// TwinCAT 3 PLC project IBF_Utilities
// Title: IBF_Utilities
// Company: Industrial Brains B.V.
// ProjectVersion: 2.0.0.0
// Description: Utilities library contains all basic utilities needed like system variables, messages, parameters etc.
// ProgramVersion: 3.1.4022.4
// libraries:
//   Tc2_Standard, * (Beckhoff Automation GmbH)
//   Tc2_System, * (Beckhoff Automation GmbH)
//   Tc2_Utilities, * (Beckhoff Automation GmbH)
//   Tc3_EventLogger, * (Beckhoff Automation GmbH)
//   Tc3_Module, * (Beckhoff Automation GmbH)
// project tree:
//   Avarage/ FB_RollingAverageLREAL.TcPOU (not stored), FB_RollingAverageTime.TcPOU, F_AverageLREAL.TcPOU, F_AverageTime.TcPOU
//   BaseFunctions/ FB_Base.TcPOU, FB_Base_WithEvent.TcPOU (not stored), FB_FunctionBase.TcPOU (not stored), FB_FunctionBase_WIthEvent.TcPOU
//   Compare/Functions/ Between.TcPOU (not stored), Between360deg.TcPOU
//   Conversion/ DegS_To_Rpm.TcPOU, DegS_To_Rpm_And_MMin.TcPOU (not stored), Grey_To_Bin.TcPOU (not stored), MMin_To_Rpm_And_DegS.TcPOU, Rpm_To_DegS.TcPOU (not stored)
//   FaultsAndMessages/Functions/ FB_EventHandler.TcPOU, Fb_FaultHandler.TcPOU (not stored), FB_OperatorMessageDisplay.TcPOU
//   General/DataTypes/ Udt_TimerBandwith.TcDUT (not stored)
//   GVLs/ DataManager.TcGVL (not stored), GVL_FixedValues.TcGVL (not stored), GVL_Message.TcGVL (not stored), GVL_Parameters.TcGVL (not stored), Sys_Variables.TcGVL
//   FaultsAndMessages/DataTypes/ E_ComponentTypes.TcTLEO (not stored), E_Locations.TcTLEO (not stored), E_MessageNumbers.TcTLEO (not stored), E_FaultTypes.TcTLEO, UDT_Fault.TcDUT
//   FaultsAndMessages/ Param_Messages.TcGVL
//   MovePathCalculations/ fAccDecCalc.TcPOU
//   Parameter/DataTypes/Old/ UDT_Parameter_1.TcDUT (not stored), Udt_ParameterRetain.TcDUT (not stored), Udt_Parameter_2.TcDUT (not stored), Udt_ParLog_Old.TcDUT (not stored)
//   Parameter/DataTypes/ Udt_ParameterId.TcDUT (not stored), Udt_Parameter.TcDUT (not stored)
//   Parameter/Functions/ FB_ParameterHandler.TcPOU (not stored), Fb_ParLogging.TcPOU, F_ParToCsvLine.TcPOU
//   PathFunctions/ F_FBNameFromPath.TcPOU, F_GetLevelFromPath.TcPOU (not stored)
//   Positions/FunctionBlocks/ FB_PositionTrigger_Old.TcPOU (not stored), FB_PositionTrigger.TcPOU (not stored)
//   Positions/Functions/ F_AccDecDistanceFromTime.TcPOU, F_AccDecDistanceFromVelo.TcPOU, F_PosCheck.TcPOU (not stored), F_TopVelocityFromTime.TcPOU, F_TriggerPosOffset.TcPOU
//   StepFunctions/ FB_CycleTrigger.TcPOU, FB_Step.TcPOU
//   System/Functions/DataManagement/ FB_PersistentDataManager.TcPOU (not stored)
//   System/Functions/ Fb_SystemVariables.TcPOU (not stored)
//   / Utilities_CD.TcCD (not stored)

// ---- FaultsAndMessages/DataTypes/E_FaultTypes.TcTLEO
{attribute 'qualified_only'}
{attribute 'strict'}
{attribute 'to_string'}
TYPE E_FaultTypes :
(
	NA	:= 0, // Not applicable
	OM 	:= 1, // Operator message
	MC	:= 2, // Missing condition
	CF	:= 3, // Cycle Fault
	FF	:= 4, // Fatal fault
	OW  := 5  // Operator warning
)UDINT;
END_TYPE

// ---- FaultsAndMessages/DataTypes/UDT_Fault.TcDUT
TYPE UDT_Fault :
STRUCT
	// active 
		Active 			: BOOL 				:= FALSE;
	// Message type
 		FaultType 		: E_FaultTypes 		:= E_FaultTypes.NA; // Type of message
	// Message Id number used for translation
		MessageNumber 	: UDINT				:= 0; // message number
		LocationNumber	: UDINT 			:= 0; // message number array ([1]= System, [2]= Module,[3]= sub module, [4]= Component)
	// Message discription
		Discription 	: STRING 			:= ''; // Message text discription in english (service personel only)
	// Location
		LocationName	: STRING			:= ''; // Location discription name
		ComponentType 	: E_ComponentTypes 	:= E_ComponentTypes.NA; // Part type discription
	// Time stamp
		StartTime		: DATE_AND_TIME 	:= DT#2020-1-1-00:00:00 ; // Time and date of message occurence
		EndTime			: DATE_AND_TIME		:= DT#2020-1-1-00:00:00 ; // Time and date of message end
	// Module number
		nModuleID		: UDINT 			; // module reference number used for fault, enable, reset, and safety functions (default := 1, 0 = main system)
	// CompleteFaultnumber for visualization
		FullFaultId		: STRING 			:= 'NA.0.0.0'; // Full fault id for use in HMI is writen by fault function [fault type, message#, location#,ComponentType]
END_STRUCT
END_TYPE

// ---- GVLs/Sys_Variables.TcGVL
(* System variables *)
{attribute 'qualified_only'}
VAR_GLOBAL
// SystemFuntion
	fbSystemVariables : Fb_SystemVariables ;
	AlwaysOn		:BOOL 			;// System variable, Always on bit
	AlwaysOff		:BOOL 			;// System variable, Always off bit
	BlinkFast		:BOOL 			;// System variable, Blink fast bit 1sec 
	BlinkSlow		:BOOL 			;// System variable, Blink slow bit 2 sec
	Pulse1Sec		:BOOL 			;// System variable, Pulse 1 cycle every second
	Pulse100ms		:BOOL 			;// System variable, pulse 1 cycle every 100 ms
	SystemTime		:DT				; // System variable, Windows system time
	TimeZoneId		:E_TimeZoneID 	; // System variable, time zone Id 
	HeartBeat		:BOOL 			;// System Variable, Main system heartbeat 0.5 sec on 0.5 sec off
END_VAR

// ---- FaultsAndMessages/Param_Messages.TcGVL
{attribute 'qualified_only'}
VAR_GLOBAL CONSTANT
	nMAX_MESSAGES_SHOWN 	: UDINT := 10 	;
	nMAX_MESSAGE_HISTORY	: UDINT := 1000 ;
	nMAX_CSV_FIELD_LENGTH	: UDINT := 100	;
	tMESSAGE_TIMEOUT		: TIME 	:= T#5S ;
	sLOGFILE_PATH			: STRING:= 'D:\FaultLogs\'	;
	sLOGFILE_NAME			: STRING:= 'Faultlog' 		; // Message log destination file
	nMESSAGE_COLUMNS		: UDINT := 8 ;
END_VAR

// ---- Avarage/FB_RollingAverageTime.TcPOU
FUNCTION_BLOCK PUBLIC FB_RollingAverageTime
VAR_INPUT
	fInputValue	: TIME ; // Input value [Anny_Number] 
END_VAR
VAR_IN_OUT
	bNewValue		: BOOL ; // Add value to array (set back to false)
	arTimeValues 	: ARRAY [*] OF TIME ; // Array of LREAL values, from thich to get the average
END_VAR
VAR_OUTPUT
	fAverage	: TIME ; // Everage of entries
END_VAR
VAR
	nWriteIndex			: DINT := 0;
	nArrayUpperBound 	: DINT;
	nArrayLowerBound 	: DINT;
	
	reNewValue	: R_TRIG ; // New value trigger
END_VAR

// determine array boundries
nArrayLowerBound := LOWER_BOUND(arTimeValues,1);
nArrayUpperBound := LOWER_BOUND(arTimeValues,1);

// Check if nwrite index is within array bounds
nWriteIndex := LIMIT(nArrayLowerBound, nWriteIndex, nArrayUpperBound);

// Add value to Array 
reNewValue(CLK := bNewValue);
IF reNewValue.Q THEN
	arTimeValues[nWriteIndex] := fInputValue;
	IF nWriteIndex = nArrayUpperBound THEN
		nWriteIndex := nArrayLowerBound;
	ELSE
		nWriteIndex := nWriteIndex +1;
	END_IF
END_IF 

// Calculate average value 
fAverage := F_AverageTime(arTimeValues);

METHOD PUBLIC Cmd_Reset : BOOL
VAR_INPUT
END_VAR
MEMSET(destAddr := ADR(arTimeValues), 0, n := SIZEOF(arTimeValues));
Cmd_Reset := true;
END_METHOD

END_FUNCTION_BLOCK

// ---- Avarage/F_AverageTime.TcPOU
FUNCTION F_AverageTime : TIME
VAR_IN_OUT
	arTimeValues : ARRAY [*] OF TIME ; // Array of LREAL values, from thich to get the average
END_VAR
VAR
	i		: DINT ;
	xSum 	: TIME ; 
	xCount	: DINT ;
END_VAR

FOR i := LOWER_BOUND(arTimeValues,1) TO UPPER_BOUND(arTimeValues,1) DO 
	xSum 	:= arTimeValues[i] + xSum;
	xCount 	:= xCount + 1 ; 
END_FOR

IF xCount >0 THEN 
	F_AverageTime := xSum / xCount;
END_IF

END_FUNCTION

// ---- Avarage/F_AverageLREAL.TcPOU
FUNCTION F_AverageLREAL : LREAL
VAR_IN_OUT
	arLREALValues : ARRAY [*] OF LREAL ; // Array of LREAL values, from thich to get the average
END_VAR
VAR
	i		: DINT ;
	xSum 	: LREAL ; 
	xCount	: DINT ;
END_VAR

FOR i := LOWER_BOUND(arLREALValues,1) TO UPPER_BOUND(arLREALValues,1) DO 
	xSum 	:= arLREALValues[i] + xSum;
	xCount 	:= xCount + 1 ; 
END_FOR

IF xCount >0 THEN 
	F_AverageLREAL := xSum / xCount;
END_IF

END_FUNCTION

// ---- BaseFunctions/FB_Base.TcPOU
FUNCTION_BLOCK PUBLIC ABSTRACT FB_Base
{attribute 'reflection'}
VAR_INPUT
	bEnable			: BOOL 		:= TRUE 	; // Module enable signal reference Default := TRUE (when using system library := GVL_Main.stModules[nModuleId].bEnabled)
	refFbParHandler	: REFERENCE TO Fb_ParLogging 	:= GVL_Parameters.fbParameterHandler	; // reference to parameter handler
	bCmdPause 		: BOOL 		:= FALSE	; // Command Pause functions		
END_VAR
VAR_IN_OUT
	refFbFault	: Fb_FaultHandler	; // reference to fault handler ( when using utilities library := GVL_Main.stModules[nModuleId].fbFaultHandler)
END_VAR
VAR_OUTPUT
	bInitOk			: BOOL 			:= FALSE 	; // function is initialized
	bBussy 			: BOOL 			:= FALSE 	; // device is busy
	bReady			: BOOL 			:= FALSE 	; // device is ready for new command 
	bErrorActive	: BOOL			:= FALSE	; // device Error active 
END_VAR
VAR
	sName			: STRING 		:= ''		; // Name of device distilled from the path 
	nLocationId		: UDINT 		:= 0		; // device id number made up of module and device number				
	
	stFault			: UDT_Fault		; // Fault data from device

	// Function path 
	{attribute 'instance-path'} 
    {attribute 'noinit'}
	sPath			: STRING	; // Path name of function (used for manual reference)
END_VAR

IF __ISVALIDREF(refFbFault) THEN 
	// check if fault is active and send to fault handler
	refFbFault.CmdAddFault(stFault);
END_IF

METHOD PUBLIC CmdReset : BOOL
VAR_INPUT
END_VAR
bErrorActive := FALSE ;

CmdReset := TRUE ;
END_METHOD

METHOD PROTECTED ExecIdentifyDevice : BOOL
VAR_INPUT
	// Message location data
	nId				: UDINT ; // Identification number of object
	nParentId		: UDINT ; // Id of higher level If aplicable (0 = no parent)
	eComponentType	: E_ComponentTypes ; // COmponent or function type for message compilation
END_VAR
// Check device ID
IF nLocationId = 0 THEN
	nLocationId := (nParentId * 10000) + nId * 100 ;
END_IF

// set message location information
stFault.ComponentType 	:= eComponentType;
stFault.LocationName	:= F_FBNameFromPath(sPath := sPath);
stFault.LocationNumber	:= nLocationId ; 

// Get device name from function and add device to manual
IF sName = '' THEN 
	sName := F_FBNameFromPath(sPath := sPath);
END_IF

ExecIdentifyDevice := nLocationId <> 0 AND sName <> '';
END_METHOD

END_FUNCTION_BLOCK

// ---- Parameter/Functions/Fb_ParLogging.TcPOU
FUNCTION_BLOCK PUBLIC Fb_ParLogging EXTENDS FB_ParameterHandler
VAR_OUTPUT
	stParLog		: Udt_ParLog_Old ; // active parameter list
	bReadBusy		: BOOL		:= FALSE	; // File acces Bussy
	bWriteBusy		: BOOL 		:= FALSE	; // file write bussy
	bError			: BOOL		:= FALSE	; // File acces error
	nErrId			: UDINT		:= 0		; // File acces error Id
	nRow	 		: UDINT 	:= 0		;(* Row number (record) *)
	nColumn			: UDINT 	:= 0		;(* Column number (record field) *)
	nInitStep		: UDINT 	:= 0 		; // Initialization step
END_VAR
VAR
	// ====== Compare array =====
		arFileParameters		: ARRAY [1..GVL_Parameters.MAX_PARAMETERS] OF Udt_Parameter;
		nNumberOfParFromFile	: UDINT; // Number of parameters read from file
		nNumberOfChanges		: UDINT; // Number of parameter changes 
		arChangeLog				: ARRAY [0..(GVL_Parameters.MAX_PARAMETERS * 2)] OF STRING ; // Parameter change log 
	// ====== Internal commands ======
		bCmdParFileWrite	: BOOL ; // write alle parameters to .csv file
		bCmdParLogWrite		: BOOL ; // write all changes to .csv file
		bCmdParFileRead		: BOOL ; // Read all parameters from .csv file 
		StParameter			: UDT_Parameter_1 ;
	// ====== File headers ======
		sCsvFileHeader : STRING := 'NUMBER;NAME;TYPE;DISCRIPTION;FACTORY;MAXIMUM;MINIMUM;UNIT;VALUE$L';
	// ====== internal status ======
		bInitOK				: BOOL 	:= FALSE ; // init has been done succesfully
		bFileNotFound		: BOOL 	:= FALSE ; // Parameter file has not been found 
		bParCountDiference	: BOOL 	:= FALSE ; // The number of parameters from file does not match machine 
		bParNumberDiference	: BOOL 	:= FALSE ; // The parameters from file do not match machine
		nDiferenceRow		: UDINT	:= 0	 ; // The file array row number in which diferences were found
 
	// ====== Current step =====
		nReadStep			: INT 	:= 0 	; // File read stepper
		nLogStep			: INT 	:= 0 	; // File logging step
		nWriteStep			: INT 	:= 0 	; // File Write stepper

	// ====== Read variables ======
		hFile				: UINT	:= 0;(* File handle of the source file *)
		cbField				: UDINT	;(* Number of bytes in field buffer *)

	// ====== Read variables ======
		sCSVLine			: T_MaxString := '';(* Single CSV text line (row, record), we are using string as record buffer (your are able to see created fields) *)
		sCSVField			: T_MaxString := '';(* Single CSV field value (column, record field) *)
		sCSVFieldString		: T_MaxString := '';// CSV field converted into string
	// ====== Functions ======
		fbFileOpenForRead	: FB_FileOpen	;(* Opens file *)
		fbFileOpenForWrite	: FB_FileOpen	;(* Opens file *)
		fbFileOpenForLog	: FB_FileOpen	;(* Opens file *)
		fbFileClose			: FB_FileClose	;(* Closes file *)
		fbFileGets			: FB_FileGets	;(* Reads one record (line) *)
		fbFilePuts			: FB_FilePuts	;(* Writes one record (line) *)
		fbReader			: FB_CSVMemBufferReader;(* Helper function block used to parse CSV data bytes (single record line) *)
		fbWriter			: FB_CSVMemBufferWriter;(* Helper function block used to create CSV data bytes (single record line) *)
	
	// Par Read timeout 
		TonParWriteTimeout	: TON := (PT := T#5S) ; // Timeout for parameter read
		TonParreadTimeout	: TON := (PT := T#5S) ; // Timeout for parameter read
		
END_VAR

SUPER^();

// ===== init =====
	IF NOT binitok THEN 
		RETURN;
	ELSE 
		CmdParWriteToFile();
		CmdParLoadFromFile();
	END_IF

METHOD PRIVATE CmdParLoadFromFile : BOOL
VAR_INPUT
END_VAR
VAR 
	i : UDINT ;
	fTempValue	: LREAL ; // Tomporary value to be placed in save value
END_VAR
IF ExecFileRead() THEN 
	;
ELSE
	RETURN;
END_IF

// Compare Parameter counters 
IF nNumberOfParameters <> nNumberOfParFromFile THEN
	bParCountDiference := TRUE ;
ELSE 
	bParCountDiference := FALSE ;
END_IF

// Compare Parameter from file with parameters in machine then write from file to machine
bParNumberDiference := FALSE ;
nDiferenceRow		:= 0 ;
IF NOT bParCountDiference THEN 
	FOR i := 1 TO nNumberOfParameters DO
		IF arParameters[i].nNumber <> arFileParameters[i].nNumber THEN
			bParNumberDiference := TRUE ;
			nDiferenceRow		:= i ;
			CONTINUE;
		ELSE
			IF (arParameters[i].pParameter^.fValue <> arFileParameters[i].fValue) THEN 
				fTempValue := arParameters[i].pParameter^.fValue;  
			ELSE
				fTempValue := 0;
			END_IF
			arParameters[i].pParameter^			:= arFileParameters[i];
			arParameters[i].pParameter^.fSaved 	:= fTempValue;
		END_IF
	END_FOR
END_IF 

CmdParLoadFromFile := TRUE ;
END_METHOD

METHOD PRIVATE CmdParWriteToFile : BOOL
VAR_INPUT
END_VAR
VAR
	i : UDINT ;
	sDTString : STRING ;
END_VAR

IF bCmdParFileWrite THEN 
	FOR i := 1 TO nNumberOfParameters DO
			// Save current actual value for later restore
			IF arParameters[i].pParameter^.fValue <> arFileParameters[i].fValue THEN
				arParameters[i].pParameter^.fSaved := arFileParameters[i].fValue ;
			END_IF
			arFileParameters[i] := arParameters[i].pParameter^ ;
	END_FOR
END_IF

//IF nNumberOfChanges > 0 AND NOT bParCountDiference THEN 
//	ExecWriteToLog();
//END_IF
CmdParWriteToFile := ExecFileWrite();
END_METHOD

METHOD PUBLIC CmdSavePar : BOOL
VAR_INPUT
END_VAR
bCmdParFileWrite := TRUE ;

CmdSavePar := bWriteBusy ;
END_METHOD

METHOD PRIVATE ExecFileRead : BOOL
VAR_INPUT
END_VAR
VAR
	i : UDINT := 0 ;
END_VAR
// ===== Wait for command =====
	IF bCmdParFileRead OR bReadBusy THEN 
		;
	ELSE
		RETURN ;
	END_IF

// ===== prepare for file read =====
	CASE nReadStep OF
		0:	(* Wait for rising edge at bRead variable *)
			bReadBusy		:= TRUE;
			bFileNotFound	:= FALSE ;
			bCmdParFileRead := FALSE ;
			bError			:= FALSE;
			nErrId			:= 0;
			hFile			:= 0;
			nRow			:= 0;
			nColumn			:= 0;
			nReadStep 			:= 1;
	
		1:	(* Open source file *)
			fbFileOpenForRead(  bExecute := FALSE  );
			fbFileOpenForRead( sNetId := GVL_Parameters.sNetId, sPathName := GVL_Parameters.sPARLIST_FILE, nMode := FOPEN_MODEREAD OR FOPEN_MODETEXT,(* Open file in text mode! *)
						ePath := PATH_GENERIC, bExecute := TRUE );
			nReadStep := 2;
	
		2:(* Wait until open not busy *)
			fbFileOpenForRead( bExecute := FALSE, bError => bError, nErrID => nErrID, hFile => hFile );
			IF NOT fbFileOpenForRead.bBusy THEN
				IF NOT fbFileOpenForRead.bError THEN
					nReadStep := 3;
				ELSE(* Error: file not found? *)
					bFileNotFound := TRUE ;
					nReadStep := 100;
				END_IF
			END_IF
		3:	(* Read single line (record) *)
			fbFileGets( bExecute := FALSE );
			fbFileGets( sNetId := GVL_Parameters.sNetId, hFile := hFile, bExecute := TRUE );
			nReadStep := 4;
		4:(* Wait until read not busy *)
			fbFileGets( bExecute := FALSE, bError => bError, nErrID => nErrID, sLine => sCSVLine );
			IF NOT fbFileGets.bBusy THEN
				IF NOT fbFileGets.bError THEN
					IF fbFileGets.bEOF THEN
						nReadStep 				:= 10;(* End of file reached => Close source file *)
					ELSE
						(* FB_FileGets returns text line without the CR (carriage return) character.
						We have to restore the CR character (replace the $L character with $R$L characters) *)
						IF RIGHT( sCSVLine, 1 ) = '$L' THEN
							sCSVLine := REPLACE( sCSVLine, '$R$L', 2, LEN( sCSVLine ) );
						END_IF
						nReadStep := 5;
					END_IF
				ELSE(* Error *)
					nReadStep := 100;
				END_IF
			END_IF
		5:(* Parse single line (record) *)
			fbReader.eCmd := eEnumCmd_First;(* Read first field value *)
			REPEAT
				fbReader( pBuffer := ADR( sCSVLine ), cbBuffer := SIZEOF( sCSVLine ), getValue => sCSVField );
				IF fbReader.bOk THEN
					fbReader.eCmd := eEnumCmd_Next;(* Read next field value *)
					IF ( nRow <= GVL_Parameters.MAX_PARAMETERS ) AND nRow > 0 THEN
						IF ( nColumn <= GVL_Parameters.PAR_COLUMNS ) THEN
							sCSVFieldString	:= CSVFIELD_TO_STRING( sCSVField, TRUE);
							CASE nColumn OF
									0: // Parameter number [Udint]	
										arFileParameters[nRow].nNumber		:= STRING_TO_UDINT(sCSVFieldString); 						
									1: // Parameter Name [string]
										arFileParameters[nRow].sName 		:= sCSVFieldString;							
									2: // Parameter type [String]
										arFileParameters[nRow].sType 		:= sCSVFieldString;	
									3: // Parameter discription [string]
										arFileParameters[nRow].sDiscription	:= sCSVFieldString;						
									4: // Parameter factory value [LREAL]
										arFileParameters[nRow].fFactory		:= STRING_TO_LREAL(sCSVFieldString);							
									5: // Parameter maximum value [LREAL]
										arFileParameters[nRow].fMaximum		:= STRING_TO_LREAL(sCSVFieldString);							
									6: // Parameter minimum value[LREAL]
										arFileParameters[nRow].fMinimum		:= STRING_TO_LREAL(sCSVFieldString);							
									7: // Parameter unit {String]
										arFileParameters[nRow].sUnit 		:= sCSVFieldString;							
									8: // Parameter value [LREAL]
										arFileParameters[nRow].fValue		:= STRING_TO_LREAL(sCSVFieldString);							
							ELSE
								;
							END_CASE
							nColumn := nColumn + 1;(* Increment number of read columns *)
						END_IF
					END_IF
					IF fbReader.bCRLF THEN(* CRLF == TRUE => End of reacord reached *)
						nNumberOfParFromFile := nRow;
						nRow 		:= nRow + 1;(* Increment number of read records *)
						nColumn 	:= 0;(* Reset number of columns *)
					END_IF
				ELSE(* Error: End of record reached or all fields read *)
					nReadStep := 3;(* Try to read next line *)
				END_IF
			UNTIL NOT fbReader.bOk
			END_REPEAT
		10:	(* Close source file *)
			fbFileClose( bExecute := FALSE );
			fbFileClose( sNetId := GVL_Parameters.sNetId, hFile := hFile, bExecute := TRUE );
			nReadStep := 11;
	
		11:(* Wait until close not busy *)
			fbFileClose( bExecute := FALSE, bError => bError, nErrID => nErrID );
			IF ( NOT fbFileClose.bBusy ) THEN
				hFile := 0;
				nReadStep := 100;
			END_IF
		100: (* Error or ready nReadStep => cleanup *)
			IF ( hFile <> 0 ) THEN
				nReadStep := 10; (* Close the source file *)
			ELSE
				bReadBusy := FALSE;
				ExecFileRead := TRUE ;
				nReadStep := 0;	(* Ready *)
			END_IF
	END_CASE
	
	TonParreadTimeout(IN := bReadBusy);
	bError S= TonParreadTimeout.Q;
END_METHOD

METHOD INTERNAL ExecFileWrite : BOOL
VAR_INPUT
END_VAR
// ===== Wait for command =====
	IF bCmdParFileWrite OR bWriteBusy THEN 
		;
	ELSE
		RETURN ;
	END_IF

// ===== Start file write =====
	CASE nWriteStep OF
		0:	(* Wait for rising edge at bWrite variable *)
				bFileNotFound		:= FALSE ;
				bParCountDiference	:= FALSE ;
				bWriteBusy 			:= TRUE;
				bCmdParFileWrite	:= FALSE ;
				bError				:= FALSE;
				nErrId				:= 0;
				hFile				:= 0;
				nRow				:= 0;
				nWriteStep 				:= 1;
		1:	(* Open source file *)
			fbFileOpenForWrite(  bExecute := FALSE  );
			fbFileOpenForWrite( sNetId := GVL_Parameters.sNetId, sPathName := GVL_Parameters.sPARLIST_FILE, nMode := FOPEN_MODEWRITE OR FOPEN_MODETEXT,(* Open file in TEXT mode! *)
						ePath := PATH_GENERIC, bExecute := TRUE );
			nWriteStep := 2;
		2:(* Wait until open not busy *)
			fbFileOpenForWrite( bExecute := FALSE, bError => bError, nErrID => nErrID, hFile => hFile );
			IF NOT fbFileOpenForWrite.bBusy THEN
				IF NOT fbFileOpenForWrite.bError THEN
					nWriteStep := 3;
				ELSE(* Error: file not found? *)
					nWriteStep := 100;
				END_IF
			END_IF
	
		3:(* Convert one PLC parameter field to CSV format *)
			// Go column by column to avoid return strings that are too long
			// TODO test (default string constructor is 80 characters, but can be extended to <?>)
			IF nRow = 0 THEN 
				sCSVLine := sCsvFileHeader;
			ELSE
				sCSVLine := F_ParToCsvLine(stParameter := arFileParameters[nRow], nColumn := nColumn);
			END_IF
			nWriteStep := 4 ;
		4:	(* Write single Field *)
			fbFilePuts( bExecute := FALSE );
			fbFilePuts( sNetId := GVL_Parameters.sNetId, hFile := hFile, sLine := sCSVLine, bExecute := TRUE );
			nWriteStep := 5;
		5:(* Wait until write not busy *)
			fbFilePuts( bExecute := FALSE, bError => bError, nErrID => nErrID );
			IF NOT fbFilePuts.bBusy THEN
				IF NOT fbFilePuts.bError THEN
					nWriteStep := 3;(* Write next record *)
					IF nRow = 0 OR nColumn = 8 THEN
						nColumn := 0 ;
						nRow := nRow + 1;
						IF nRow = nNumberOfParameters + 1 THEN
							nWriteStep := 10;
						END_IF;
					ELSE
						nColumn := nColumn + 1;
					END_IF
				ELSE(* Error *)
					nWriteStep := 100;
				END_IF
			END_IF
		10:	(* Close source file *)
			fbFileClose( bExecute := FALSE );
			fbFileClose( sNetId := GVL_Parameters.sNetId, hFile := hFile, bExecute := TRUE );
			nWriteStep := 11;
	
		11:(* Wait until close not busy *)
			fbFileClose( bExecute := FALSE, bError => bError, nErrID => nErrID );
			IF ( NOT fbFileClose.bBusy ) THEN
				hFile := 0;
				nWriteStep := 100;
			END_IF
	
		100: (* Error or ready nWriteStep => cleanup *)
			IF ( hFile <> 0 ) THEN
				nWriteStep := 10; (* Close the source file *)
			ELSE
				bParCountDiference 	:= FALSE ;
				bWriteBusy 			:= FALSE;
				ExecFileWrite		:= TRUE ;
				nWriteStep 			:= 0;	(* Ready *)
			END_IF
	
	END_CASE
	
	TonParWriteTimeout(IN := bWriteBusy);
	bError	S= TonParWriteTimeout.Q ;
	

ExecFileWrite := TRUE ;
END_METHOD

METHOD PRIVATE ExecWriteToLog : BOOL
VAR_INPUT
END_VAR
VAR
	sTempField : STRING ;
END_VAR
// ===== Wait for command =====
	IF bWriteBusy OR bCmdParLogWrite THEN 
		;
	ELSE
		RETURN ;
	END_IF

// ===== Start file write =====
CASE nLogStep OF
	0:	(* Wait for rising edge at bWrite variable *)
			bWriteBusy 			:= TRUE;
			bCmdParLogWrite	:= FALSE ;
			bError				:= FALSE;
			nErrId				:= 0;
			hFile				:= 0;
			nRow				:= nNumberOfChanges * 2; // Twice the number of changes because old and new values are stored sequentially in teh same array
			nLogStep 			:= 1;
	1:	(* Open source file *)
		fbFileOpenForLog(  bExecute := FALSE  );
		fbFileOpenForLog( sNetId := GVL_Parameters.sNetId, sPathName := GVL_Parameters.sPARLIST_FILE, nMode := FOPEN_MODETEXT,(* Open file in TEXT mode! *)
					ePath := PATH_GENERIC, bExecute := TRUE );
		nLogStep := 2;
	2:(* Wait until open not busy *)
		fbFileOpenForLog( bExecute := FALSE, bError => bError, nErrID => nErrID, hFile => hFile );
		IF NOT fbFileOpenForLog.bBusy THEN
			IF NOT fbFileOpenForLog.bError THEN
				nLogStep := 3;
			ELSE(* Error: file not found? *)
				nLogStep := 100;
			END_IF
		END_IF

	3:(* Convert one PLC record to CSV format *)
		sCSVLine := arChangeLog[nRow];
		nLogStep := 4 ;
	4:	(* Write single text line *)
		fbFilePuts( bExecute := FALSE );
		fbFilePuts( sNetId := GVL_Parameters.sNetId, hFile := hFile, sLine := sCSVLine, bExecute := TRUE );
		nLogStep := 5;

	5:(* Wait until write not busy *)
		fbFilePuts( bExecute := FALSE, bError => bError, nErrID => nErrID );
		IF NOT fbFilePuts.bBusy THEN
			IF nRow = 0 THEN
				nNumberOfChanges := 0;
				nLogStep := 10;
			ELSIF NOT fbFilePuts.bError THEN
				arChangeLog[nRow] := ''; // Delete change from log
				nRow := nRow - 1;
				nLogStep := 3;(* Write next record *)
			ELSE(* Error *)
				nLogStep := 100;
			END_IF
		END_IF
	10:	(* Close source file *)
		fbFileClose( bExecute := FALSE );
		fbFileClose( sNetId := GVL_Parameters.sNetId, hFile := hFile, bExecute := TRUE );
		nLogStep := 11;

	11:(* Wait until close not busy *)
		fbFileClose( bExecute := FALSE, bError => bError, nErrID => nErrID );
		IF ( NOT fbFileClose.bBusy ) THEN
			hFile := 0;
			nLogStep := 100;
		END_IF

	100: (* Error or ready nLogStep => cleanup *)
		IF ( hFile <> 0 ) THEN
			nLogStep := 10; (* Close the source file *)
		ELSE
			bWriteBusy := FALSE;
			nLogStep := 0;	(* Ready *)
		END_IF
END_CASE
END_METHOD

METHOD PUBLIC Init : BOOL
VAR_INPUT
END_VAR
// Read parameters from .CSV file and check if load is valid

CASE nInitStep OF 
	0: //check if init has been done 
		bInitOK 	:= FALSE;
		nInitStep 	:= 10 ;
	10: // start File read
		bCmdParFileRead := TRUE ;
		nInitStep := 11; 
	11: // Execute file read 
		IF CmdParLoadFromFile() THEN 
			nInitStep := 12 ;
		END_IF
	12: // Check if read is valid 
		IF bFileNotFound OR bParCountDiference THEN 
			nInitStep := 20 ;
		ELSE 
			nInitStep := 100 ;
		END_IF
	20: // start File write
		bCmdParFileWrite:= TRUE ;
		nInitStep		:= 21 ;
	21: // Wait for file write to finish
		IF CmdParWriteToFile() THEN 
			nInitStep := 100 ;
		ELSIF bError THEN 
			nInitStep := 900 ; 
		END_IF 
	100: // Init ok 
		bInitOK 	:= TRUE ;
		Init		:= TRUE ;
		nInitStep	:= 0 ;
	900: // file fault	
		bInitOK := FALSE ;
		RETURN ;
	ELSE 
		;
END_CASE
END_METHOD

END_FUNCTION_BLOCK

// ---- Parameter/Functions/F_ParToCsvLine.TcPOU
FUNCTION F_ParToCsvLine : T_MaxString // convert parameter into csv string (default UDt_Parameter setup)
VAR_INPUT
	stParameter : Udt_Parameter ; 
	nColumn		: UDINT ;
END_VAR
VAR
	sTempString : T_MaxString;
	sTempCsvField : T_MaxString;
END_VAR

CASE nColumn OF 
	0: // number
		sTempString := UDINT_TO_STRING(stParameter.nNumber);
	1: // name
		sTempString := stParameter.sName;
	2: // Type
		sTempString := stParameter.sType;
	3: // discription
		sTempString := stParameter.sDiscription;
	4: // factory
		sTempString := LREAL_TO_STRING(stParameter.fFactory);
	5: // maximum
		sTempString := LREAL_TO_STRING(stParameter.fMaximum);
	6: // minimum
		sTempString := LREAL_TO_STRING(stParameter.fMinimum);
	7: // Unit 
		sTempString := stParameter.sUnit;
	8: // value
		sTempString := LREAL_TO_STRING(stParameter.fValue);
	ELSE
		;
END_CASE

sTempCsvField := STRING_TO_CSVFIELD(sTempString, FALSE);
IF nColumn < 8 THEN 
	sTempCsvField := CONCAT(StempCsvField,';');
ELSE
	sTempCsvField := CONCAT(StempCsvField,'$L');
END_IF

F_ParToCsvLine := sTempCsvField;

END_FUNCTION

// ---- PathFunctions/F_FBNameFromPath.TcPOU
FUNCTION F_FBNameFromPath : STRING // distills .fb name from function path
VAR_INPUT
	sPath	: STRING ;
END_VAR
VAR
	sTemp		: STRING ;
	nstartFbName: INT ; 
END_VAR

sTemp := sPath ;

REPEAT 
	// Look for first occurance of .fb in string
	nStartFbName := FIND( sTemp,'.fb');
	// Delete text before .fb and .fb itself
	IF nstartFbName <>0 THEN 
		sTemp := DELETE( STR := sTemp, LEN := nstartFbName + 3, 0); 
	END_IF
UNTIL
	nstartFbName = 0 
END_REPEAT

F_FBNameFromPath := sTemp ;

END_FUNCTION

// ---- BaseFunctions/FB_FunctionBase_WIthEvent.TcPOU
{attribute 'reflection'}
FUNCTION_BLOCK PUBLIC ABSTRACT FB_FunctionBase_WIthEvent EXTENDS FB_Base_WithEvent
VAR_INPUT
	bSafetyOk	: BOOL 		:= TRUE 				; // Module can operate safely [default true]
END_VAR
VAR_OUTPUT
	sActiveState	: STRING 		:= 'Idle'	; // active state of device 
	bManual			: BOOL 			:= FALSE 	; // device is in manual mode
	bIsSafe			: BOOL 			:= FALSE	; // Device is locked and safe
	bHeld			: BOOL 			:= FALSE 	; // Function is held
	bBlockedCommand	: BOOL 			:= FALSE 	; // a device command is blocked because of collision detect 
END_VAR
VAR
	bCmdManual 		: BOOL			:= FALSE	; // manual commands enabled control functions (thus disable automatic)
END_VAR

SUPER^();

// Communicate active state
IF NOT bSafetyOk THEN 
	sActiveState := 'Safety not ok';
ELSIF bErrorActive THEN 
	sActiveState := 'Error is active';
ELSIF NOT bInitOk THEN 
	sActiveState := 'Not initialized';
ELSIF bManual THEN 
	sActiveState := 'Operational';
END_IF 

// check for manual command mode
bManual := bCmdManual ;

// Execute device functions
IF bInitOk THEN  
	ExecMachineSafety();
	ExecDevFunctions();
END_IF

// Set fault if commands are blocked
IF bBlockedCommand THEN 
	fbEvent.CmdAddEvent( Event := TC_EVENTS.StateMessages.FunctionsIsBlocked);
END_IF

METHOD PUBLIC CmdHold : BOOL
VAR_INPUT
END_VAR
bHeld 	:= TRUE ;
CmdHold := bHeld ;
END_METHOD

METHOD PUBLIC CmdManual : BOOL
VAR_INPUT
END_VAR
bCmdManual := true ;
END_METHOD

METHOD PUBLIC CmdSafeStop : BOOL
VAR_INPUT
END_VAR
// check if device is safe
bIsSafe 	:= NOT bEnable ;
CmdSafeStop := bIsSafe ;
END_METHOD

METHOD PROTECTED ExecDevFunctions : BOOL
VAR_INPUT
END_VAR
END_METHOD

METHOD PROTECTED ExecMachineSafety : BOOL
VAR_INPUT
END_VAR
END_METHOD

END_FUNCTION_BLOCK

// ---- Compare/Functions/Between360deg.TcPOU
FUNCTION Between360deg : BOOL // Returns true if value is >= the lower and <= the upper threshold, if lower > upper then upper := Upper +360 deg
VAR_INPUT
	Lower	: LREAL	; // lower threshold value [LREAL]
	Value	: LREAL	; // test value [LREAL]
	Upper	: LREAL	; // Upper threshold value [LREAL]
END_VAR
VAR
END_VAR

IF Lower > Upper THEN  
	Between360deg S= Between( Lower, Value, 360);
	Between360deg S= Between( 0, Value, Upper)	;
ELSE 
	Between360deg S= Between( Lower, Value, Upper)	;
END_IF

END_FUNCTION

// ---- Conversion/DegS_To_Rpm.TcPOU
(* convert degrees per second to rotations per minute *)
FUNCTION DegS_To_Rpm : LREAL
VAR_INPUT
	DegS : LREAL ; // Input degrees per second as long real
END_VAR

// ===== convert degrees per second to Rpm =====
	DegS_To_Rpm := (DegS/360)*60 ;

END_FUNCTION

// ---- Conversion/MMin_To_Rpm_And_DegS.TcPOU
(* Convert meters per minute to degrees per second *)
FUNCTION MMin_To_Rpm_And_DegS : BOOL
VAR_INPUT
	MeterPerMinute 	: LREAL ; // Input meters per minute
	StitchLength	: LREAL ; // Input Stitch length
END_VAR
VAR_OUTPUT
	RevPerMinute	: LREAL ; // Output revolutions per minute
	DegPerSecond	: LREAL ; // Output degrees per second
END_VAR
VAR
	MmMin 	: LREAL ; // Millimeters per minute
	RevSec 	: LREAL ; // Millimeters per second
END_VAR

// ===== convert MMin to RPM =====
	RevPerMinute := (MeterPerMinute * 1000) / StitchLength ;
//===== Convert RPM to DegS =====
	DegPerSecond := (RevPerMinute/60)*360 ;

END_FUNCTION

// ---- FaultsAndMessages/Functions/FB_EventHandler.TcPOU
FUNCTION_BLOCK PUBLIC FB_EventHandler
VAR_INPUT
	nTwincErrorId	: UDINT := 0; // OPTIONAL Error Id from twincat function block library
END_VAR
VAR_OUTPUT
	// Active events
	bActOM 			: BOOL := FALSE ;
	bActMC 			: BOOL := FALSE ;
	bActCF 			: BOOL := FALSE ;
	bActFF 			: BOOL := FALSE ;
	// Last event
	stLastEvent		: TcEventEntry 	; // Event entry discription  
END_VAR
VAR // Event Conformation data
	bConfRequired 	: BOOL := FALSE ; // Conformation of  		
	// Resetting
	bResetting		: BOOL := FALSE ;
END_VAR
VAR // location data
	// Location
	nLocationNumber	: UDINT 			:= 0; // message number array ([1]= System, [2]= Module,[3]= sub module, [4]= Component)
	sLocationName	: STRING			:= ''; // Location discription name
	eComponentType 	: E_ComponentTypes 	:= E_ComponentTypes.NA; // Part type discription
	// Module number
	nModuleID		: UDINT 			; // module reference number used for fault, enable, reset, and safety functions (default := 1, 0 = main system)
	// Source
	fbSource		: FB_TcSourceInfo;
END_VAR
VAR // Event functions 
	fbAlarm		: FB_TcAlarm ; // alarm event function
	fbMessage 	: FB_TcMessage ; // Message event
	
	hr 			: HRESULT;
	hrLastError : HRESULT;
END_VAR

METHOD PUBLIC CmdAddEvent : BOOL
VAR_INPUT
	Event			: TcEventEntry ; // Event entry discription  
END_VAR
// check if allarm has already been raised
IF fbAlarm.EqualsToEventEntryEx(stOther	:= Event) THEN
	CmdAddEvent := TRUE;
	RETURN;
END_IF

// Check Event severity
CASE Event.eSeverity OF 
	TcEventSeverity.Critical:
		bActFF 			S= TRUE ;	
		fbAlarm.CreateEx(Event,TRUE,fbSource);
		hr := fbAlarm.Raise(0);
	TcEventSeverity.Error:
		bActCF 			S= TRUE ;	
		fbAlarm.CreateEx(Event,TRUE,fbSource);
		hr := fbAlarm.Raise(0);
	TcEventSeverity.Warning:
		bActMC 			S= TRUE ;	
		fbAlarm.CreateEx(Event,FALSE,fbSource);
		hr := fbAlarm.Raise(0);
	TcEventSeverity.Info:
		bActOM 			S= TRUE ;	
		fbMessage.CreateEx(Event,fbSource);
		hr := fbMessage.Send(0);
	ELSE 
		RETURN;
END_CASE

// Add aditional error id
IF nTwincErrorId >0 THEN 
	fbAlarm.ipArguments.AddUDInt( value := nTwincErrorId);
END_IF
nTwincErrorId := 0; // Always clear error id after check

IF FAILED(hr) THEN 
	hrLastError := hr ;
ELSE
	CmdAddEvent := TRUE;
END_IF
END_METHOD

METHOD PUBLIC CmdReset : BOOL
VAR_INPUT
END_VAR
bResetting := TRUE ;

hr := fbAlarm.Clear(0,TRUE);

IF NOT FAILED(hr) THEN 
	bResetting := FALSE ; 
	bActOM 	:= FALSE ;
	bActMC	:= FALSE ;
	bActCF	:= FALSE ;
	bActFF	:= FALSE ;
END_IF

// Set feedback
CmdReset := NOT bResetting;
END_METHOD

METHOD PRIVATE ExecSetActiveEvents : BOOL
VAR_INPUT
END_VAR
END_METHOD

METHOD PUBLIC Init : BOOL
VAR_INPUT
	// Location
		sLocationName	: STRING			:= ''; // Location discription name
		eComponentType 	: E_ComponentTypes 	:= E_ComponentTypes.NA; // Part type discription
	// Module number
		nModuleID		: UDINT 			; // module reference number used for fault, enable, reset, and safety functions (default := 1, 0 = main system)
END_VAR
// Transfer location data into event location data format
fbSource.nId 	:= nModuleID;
fbSource.sName	:= TO_STRING(eComponentType);
fbSource.ExtendName(sLocationName);

fbMessage.CreateEx(TC_EVENTS.StateMessages.ModuleInitialized,fbSource);
fbMessage.Send(0);

Init := TRUE ;
END_METHOD

END_FUNCTION_BLOCK

// ---- FaultsAndMessages/Functions/FB_OperatorMessageDisplay.TcPOU
FUNCTION_BLOCK FB_OperatorMessageDisplay // function compares messages and shows latest message on screen for a set period of time
VAR_INPUT
	bEnable 	: BOOL 	:= TRUE ; // enable messages
	tDisplayTime: TIME	:= Param_Messages.tMESSAGE_TIMEOUT ; // Time before message relevance is checked (default = Param_Messages.tMESSAGE_TIMEOUT)
END_VAR
VAR_IN_OUT
	sMessage 	: STRING ; // Operator message (default = GVL_Message.sOPeratorMessage)
END_VAR
VAR_OUTPUT
	sOutMessage : STRING ; // message output to screen
END_VAR
VAR
	sOldMessage 	: STRING := ''; // old message as displayed 
	tonDisplayTimer	: TON ; // Display timer
END_VAR

// Run timers
tonDisplayTimer(PT := tDisplayTime);

// compare old message with new message 
IF sMessage = sOldMessage THEN 
	tonDisplayTimer.IN := TRUE ;
	IF tonDisplayTimer.Q = TRUE THEN 
		sMessage := '';
	END_IF
ELSE 
	tonDisplayTimer.IN 	:= FALSE 	;
	sOldMessage 		:= sMessage ; 
END_IF

// write message to display
sOutMessage := sMessage ;

END_FUNCTION_BLOCK

// ---- MovePathCalculations/fAccDecCalc.TcPOU
FUNCTION fAccDecCalc : LREAL // calculates acceleration and deceleration values from path [units/sec^2]
VAR_INPUT
	fVelocity		: LREAL ; // current velocity [units]
	fNewVelocity	: LREAL ; // New velocity [units] 
	fDistance		: LREAL ; // Travel distance [units]
END_VAR
VAR
	xDeltaVelo		: LREAL ; // delta velocity
	xAverageVelo	: LREAL ; // Average velocity
	xTime			: LREAL ; // Time it takes to slow down [s]
END_VAR

xDeltaVelo	:= ABS(fVelocity - fNewVelocity);
xAverageVelo:= ABS(fVelocity + fNewVelocity)/2;
xTime		:= fDistance / xAverageVelo ;
fAccDecCalc	:= xDeltaVelo / xTime ;

END_FUNCTION

// ---- Positions/Functions/F_AccDecDistanceFromTime.TcPOU
FUNCTION F_AccDecDistanceFromTime : LREAL
VAR_INPUT
	nAccelDecel	: LREAL ; // acceleration or deceleration [units/s^2]
	nTimeMs		: LREAL	; // Time for acceleratio/ deceleration to take place [ms]
END_VAR
VAR
	nTimeSec	: LREAL;
	nVelocity	: LREAL;
END_VAR

nTimeSec := nTimeMs/1000;

nVelocity := nAccelDecel * nTimeSec;

F_AccDecDistanceFromTime := nVelocity * nTimeSec / 2 ;

END_FUNCTION

// ---- Positions/Functions/F_AccDecDistanceFromVelo.TcPOU
FUNCTION F_AccDecDistanceFromVelo : LREAL
VAR_INPUT
	nVelocity	: LREAL ; // velocity [m/s]
	nAccDecc	: LREAL ; // acceleration or deceleration value [m/s^2]
END_VAR
VAR
	nTime : LREAL ;
END_VAR

nTime := nVelocity	/	nAccDecc ;

F_AccDecDistanceFromVelo := nVelocity * (nTime/2);

END_FUNCTION

// ---- Positions/Functions/F_TopVelocityFromTime.TcPOU
FUNCTION F_TopVelocityFromTime : LREAL
VAR_INPUT
	nAccel	: LREAL ; // acceleration or deceleration [units/s^2]
	nTimeMs		: LREAL	; // Time for acceleratio/ deceleration to take place [ms]
END_VAR
VAR
	nTimeSec	: LREAL;
END_VAR

nTimeSec := nTimeMs/1000;

F_TopVelocityFromTime := nAccel * nTimeSec;

END_FUNCTION

// ---- Positions/Functions/F_TriggerPosOffset.TcPOU
(* function to calculate trigger points for time based moves *)
FUNCTION F_TriggerPosOffset : LREAL
VAR_INPUT
	Velocity		: LREAL	; // [Units/sec] command velocity 
	nMoveTimeMs		: LREAL	; // [ms] Time it takes for move to complete
END_VAR
VAR
END_VAR

// ===== Convert time to usable calculation value =====
	F_TriggerPosOffset := nMovetimeMs * ABS(Velocity / 1000);

END_FUNCTION

// ---- StepFunctions/FB_CycleTrigger.TcPOU
FUNCTION_BLOCK FB_CycleTrigger // This function can be used to start state machines and wait for them to finish
VAR_OUTPUT
	bStart 	: BOOL ; // Start cycle 
	bBusy 	: BOOL ; // cycle is bussy
	bDone	: BOOL ; // cycle is done
END_VAR
VAR
	fbreStartCycle : R_TRIG ; // rising edge trigger for cycle start
END_VAR

ACTION Reset:
bDone 	:= FALSE;
bBusy 	:= FALSE;
bStart	:= FALSE;
END_ACTION

ACTION SetDone:
bBusy := FALSE 	;
bDone := TRUE	;
END_ACTION

ACTION SetStart:
IF fbreStartCycle.Q THEN
	bBusy := TRUE; 
ELSIF bDone THEN 
	bStart := FALSE;
ELSE
	bStart := TRUE;
END_IF

fbreStartCycle(CLK := bStart);
END_ACTION

END_FUNCTION_BLOCK

// ---- StepFunctions/FB_Step.TcPOU
FUNCTION_BLOCK PUBLIC FB_Step EXTENDS FB_Base
VAR_INPUT
END_VAR
VAR_OUTPUT
	nActStep	: UDINT := 0 ; // Active step
	bIdle		: BOOL	:= TRUE  ; // Stepper is idle (Step 0)
	bPaused		: BOOL 	:= FALSE ; // Stepper is paused
	bHold		: BOOL 	:= FALSE ; // Stepper is blocked for changes
	bSkipPause	: BOOL	:= FALSE ; // Pause function is skipped in this step 
	bResetting	: BOOL  := False ; // Reset is active
END_VAR
VAR
	nPreviousStep 	: UDINT ; // Previous active step
	nNextStep		: UDINT ; // Next step to activate
	nResetStep		: UDINT ; // step to which the stepper will go after reset
END_VAR

SetActiveStep();

METHOD PUBLIC CmdHold : BOOL
VAR_INPUT
END_VAR
bHold := TRUE ;

CmdHold := bHold;
END_METHOD

METHOD PUBLIC CmdNext : BOOL
VAR_INPUT
END_VAR
IF NOT bHold THEN 
	nNextStep := nActStep +	1 ;	
END_IF

CmdNext := TRUE ;
END_METHOD

METHOD PUBLIC CmdPrevious : BOOL
VAR_INPUT
END_VAR
IF NOT bHold THEN 
	nNextStep := nPreviousStep ;	
END_IF

CmdPrevious := TRUE ;
END_METHOD

METHOD PUBLIC CmdReset : BOOL
VAR_INPUT
END_VAR
bErrorActive := FALSE ;

IF nActStep <> nResetStep THEN 
	IF NOT bResetting THEN
		bResetting := TRUE ;
	ELSE
		nPreviousStep 	:= nActStep ;
		nNextStep		:= nResetStep ;
		nActStep 		:= nResetStep ;
		bResetting 		:= FALSE;
	END_IF
ELSE
	CmdReset := TRUE ; 
END_IF
END_METHOD

METHOD PUBLIC CmdToStep : BOOL
VAR_INPUT
	nStep	: UDINT ;
END_VAR
IF NOT bHold THEN 
	nNextStep := nStep ;
END_IF

CmdToStep := nNextStep = nStep ;
END_METHOD

METHOD PUBLIC Init : BOOL
VAR_INPUT
	// Location data for messages  
	nId			: UDINT ; // Identification number of object
	nParentId	: UDINT ; // Id of higher level If aplicable (0 = no parent)
	nResetStep	: UDINT ; // step to which the stepper wil go at reset
END_VAR
// ====== Calculate device id =====
	ExecIdentifyDevice(nId,nParentId,E_ComponentTypes.StepProgram);
	
// ===== set reset step ======
	nActStep 			:= nResetStep ;
	THIS^.nResetStep	:= nResetStep ;
END_METHOD

METHOD PRIVATE SetActiveStep : BOOL
VAR_INPUT
END_VAR
IF bResetting THEN 
	nPreviousStep 	:= nActStep ;
	nNextStep		:= nResetStep ;
	nActStep 		:= nResetStep ;
	bResetting 		:= FALSE; 
ELSIF bHold THEN 
	bHold 			:= FALSE ;
	RETURN; 
ELSIF bErrorActive THEN 
	stFault.Active			:= TRUE ;
	stFault.ComponentType	:= E_ComponentTypes.StepProgram ;
	stFault.Discription		:= CONCAT(sName, ' Invalid step state');
	stFault.FaultType		:= E_FaultTypes.FF;
	stFault.MessageNumber	:= E_MessageNumbers.FF_ComunicationFault;
ELSIF NOT bCmdPause OR bSkipPause THEN 
	IF nActStep <> nNextStep THEN 
		nPreviousStep 	:=	nActStep;	
		nActStep		:= 	nNextStep;
	END_IF
END_IF

bPaused 	:= bCmdPause ;	
bSkipPause 	:= FALSE ; 
bIdle 		:= nActStep = 0 ;
END_METHOD

METHOD Public SkipPause : BOOL
VAR_INPUT
END_VAR
bSkipPause := TRUE ;

SkipPause := true ;
END_METHOD

METHOD PUBLIC StepError : BOOL
VAR_INPUT
END_VAR
bErrorActive := TRUE ;
END_METHOD

END_FUNCTION_BLOCK
